Staubli VAL3: isLoggedIn.pgx

public program isLoggedIn(num x_nCamID (dimensions=1), bool& x_bLoggedIn (dimensions=1))
  local num l_nError
  local bool l_bOnline
begin
  //-----------------------------------------------------------------------
  //Header begin
  //Description of program
  // This routines checks wether or not we are still logged into the camera.
  // Please note that this function should not be called before loging in.
  // It is only designed to report a connection loss during read/write operations.
  //
  // Input Parameters
  //  x_nCamID :
  //    role : camera's ID
  //
  // Output Parameteres
  //  x_bLoggedIn  :
  //    role : returns true if we are logged in and false otherwise.
  //
  //Examples
  //  call isLoggedIn(nCamID,l_bLoggedIn)
  //
  //Header end
  //History
  //  Creation : 06-2012 - T.Caille - C.Rocchini
  //Header end
  //-----------------------------------------------------------------------
  call getOnline(x_nCamID,l_bOnline)
  call getErrorCode(x_nCamID,l_nError)
  x_bLoggedIn=l_nError!=202
  if !x_bLoggedIn
    cCamera[x_nCamID].bConnected=false
  endIf
end
